INTERFACE I_MqttDeviceDiscovery

METHOD DeleteDevice : BOOL
VAR_INPUT
END_VAR
END_METHOD

PROPERTY DeviceInformation : ST_MqttDeviceInformation
GET
END_GET
END_PROPERTY

PROPERTY NodeId : STRING(20)
GET
END_GET
END_PROPERTY

PROPERTY ObjectId : STRING(40)
GET
END_GET
END_PROPERTY

METHOD RegisterDevice : BOOL
VAR_INPUT
END_VAR
END_METHOD

END_INTERFACE

(* stored: Version 1.1.0.1, ProductVersion 3.1.4024.5
   Itf I_MqttDeviceDiscovery: Id {e93832ea-e390-40fa-bb33-fa8bb210e5a8}
   Method DeleteDevice: Id {37973996-03e6-4298-a383-ed456bdc262d}
   Property DeviceInformation: Id {d021716b-b41a-4219-b4ab-fb7754fbca75}
   Get Get: Id {a7f7d274-1961-4138-8036-fddcee753d61}
   Property NodeId: Id {ddb3980d-920c-48a3-8782-afcba888d87a}
   Get Get: Id {51407675-11c5-4ad3-ade9-37dc3a049507}
   Property ObjectId: Id {aec62e32-12bc-49fe-8daf-9b2e35fc352a}
   Get Get: Id {05c6a9aa-cc09-4751-a299-4a6213338543}
   Method RegisterDevice: Id {eabaaa50-efc6-4c24-bc93-e68d8b58d71a} *)
